# B&R Automation Studio project mappCnc
Automation Studio 4.12.11.2 SP; technology packages: mappCockpit 5.24.4, mappMotion 5.31.3, mappView 5.24.8

## Configuration Config1

CPU X20CP3585, AutomationRuntime U4.93, Build 4.1.2, Safety 0.0, Vc V4.73.5

CPU X20CP3684, AutomationRuntime 6.7.6, Build 11.3.0, Vc 6.7.0

### Task classes (Cpu.sw)
```
Cyclic#1:
  Cnc <- Motion.Cnc.prg
Cyclic#4 (cycle 200000 us, tolerance 200000 us):
  Draw <- Visualization.Draw.prg
DataObjects: McAcpSys
NcDataObjects: McDriveLog, World <- Motion.World.dob
VcDataObjects: Visu <- Visualization.Visu.dob
Binaries: arsvcreg, udbdef, McAcpDrv, McMechSys, McAcpSim, TCData, vcchspot, vcfile, arial, vctcal, vccbmp, vccstr, vcbclass, mCoWebSc, vcgclass, vcdsint, vcnet, vcmgr, arflatprv, Visu03, vcshared, vcrt, vcpdvnc, arcoal, vcpdsw, visvc, vcpfar00, vcctext, Visu01, vcfntttf, vcalarm, vcpkat, Visu02, vcdsloc, mvLoader, Role, iomap, Config_2, Hierarchy, Config_3, arconfig, asfw, sysconf, Config_4, User, ashwac, Config_1, ashwd, TraceConfi, Settings
Libraries: McBase, McAxGroup, McPathGen, McAxis, McProgInt, McAcpAx, MpCnc, MpBase, MpAxis, visapi, CoTrace, AsZip, FileIO, runtime, MpWebXs, AsArSdm, powerlnk, asarlog, asieccon, asmem, brsystem, astime, sys_lib, asarprof, dataobj, vcresman, arssl, asio, asepl
```

### Task classes (Cpu.sw)
```
Cyclic#1:
  Cnc <- Motion.Cnc.prg
Cyclic#4 (cycle 200000 us, tolerance 200000 us):
  Draw <- Visualization.Draw.prg
DataObjects: McAcpSys
NcDataObjects: McDriveLog, World <- Motion.World.dob
VcDataObjects: Visu <- Visualization.Visu.dob
Binaries: arsvcreg, udbdef, McAcpDrv, McMechSys, McAcpSim, TCData, vcchspot, vcfile, arial, vctcal, vccbmp, vccstr, vcbclass, mCoWebSc, vcgclass, vcdsint, vcnet, vcmgr, arflatprv, Visu03, vcshared, vcrt, vcpdvnc, arcoal, vcpdsw, visvc, vcpfar00, vcctext, Visu01, vcfntttf, vcalarm, vcpkat, Visu02, vcdsloc, mvLoader, Role, iomap, Config_2, Hierarchy, Config_3, arconfig, asfw, sysconf, Config_4, User, ashwac, Config_1, ashwd, TraceConfi, Settings
Libraries: visapi, AsZip, FileIO, runtime, AsArSdm, powerlnk, asarlog, asieccon, asmem, brsystem, astime, sys_lib, asarprof, dataobj, vcresman, arssl, asio, asepl, McBase, MpBase, McAxGroup, McAcpAx, McAxis, McPathGen, MpAxis, McProgInt, MpCnc, CoTrace
```

### Hardware
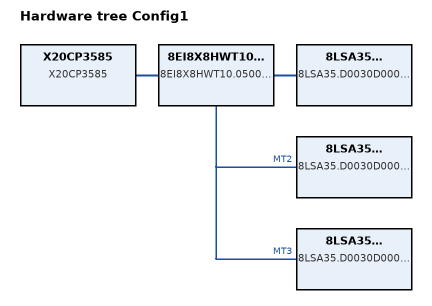
```
8EI8X8HWT10.0500-1 : 8EI8X8HWT10.0500-1 v2.4.0.0  [PLK1 -> X20CP3585.IF3 [Cable Type=PowerlinkCable, Length=10, Version=1.0.0.3]; MT2 -> 8LSA35.D0030D000-0a.MT; MT3 -> 8LSA35.D0030D000-0b.MT]
  DriveConfiguration/Module:
    McAcoposTypeID = AcoposP3TConfig
    ActivateACOPOSSimulationOnPLC = 0
  DriveConfiguration/Channel[1]/RealAxis:
    AxisReference = gAxisQX
    MechanicalElementsIsInvisible = 0
  DriveConfiguration/Channel[1]/RealAxis/MechanicalElements/Gearbox:
    InputIsReadOnly = 0
    Input = 1
    OutputIsReadOnly = 0
    Output = 1
  DriveConfiguration/Channel[1]/RealAxis/MechanicalElements/RotaryToLinearTransformation:
    ReferenceDistanceIsReadOnly = 0
    ReferenceDistance = 1
  DriveConfiguration/Channel[1]/RealAxis/EncoderLink:
    ParameterSetSelection = Automatic
  DriveConfiguration/Channel[1]/RealAxis/Controller:
    ModeIsReadOnly = 0
    Mode = PositionController
  DriveConfiguration/Channel[1]/RealAxis/Controller/Mode/Position:
    ProportionalGain = 50.0
    IntegrationTime = 0.0
    PredictionTime = 0.0004
    TotalDelayTime = 0.0004
  DriveConfiguration/Channel[1]/RealAxis/Controller/Mode/Speed:
    ProportionalGainIsReadOnly = 0
    ProportionalGain = 2.0
    IntegrationTimeIsReadOnly = 0
    IntegrationTime = 0.0
    FilterTimeIsReadOnly = 0
    FilterTime = 0.0
  DriveConfiguration/Channel[1]/RealAxis/Controller/Mode/LoopFilters:
    LoopFilterXIsReadOnly = 0
    LoopFilter1 = NotUsed
    LoopFilter2 = NotUsed
    LoopFilter3 = NotUsed
  DriveConfiguration/Channel[1]/RealAxis/Homing:
    ModeIsReadOnly = 0
    Mode = Direct
  DriveConfiguration/Channel[1]/RealAxis/Homing/Mode:
    Position = 0.0
    ReferencePulse = NotUsed
  DriveConfiguration/Channel[1]/RealAxis/Homing:
    RestorePositionVariable = 
  DriveConfiguration/Channel[1]/RealAxis/StopReaction:
    QuickstopIsReadOnly = 0
    Quickstop = DecelerationLimit
    DriveErrorIsReadOnly = 0
    DriveError = DecelerationLimit
  DriveConfiguration/Channel[1]/RealAxis/MovementErrorLimits:
    PositionError = 1.0
    VelocityErrorMonitoring = Automatic1
  DriveConfiguration/Channel[1]/RealAxis:
    JerkFilterIsReadOnly = 0
    JerkFilter = NotUsed
    ZeroVibrationFilter = NotUsed
  DriveConfiguration/Channel[1]/RealAxis/DigitalInputs/HomingSwitch:
    SourceIsReadOnly = 0
    Source = NotUsed
    Level = High
  DriveConfiguration/Channel[1]/RealAxis/DigitalInputs/PositiveLimitSwitch:
    SourceIsReadOnly = 0
    Source = NotUsed
    Level = High
  DriveConfiguration/Channel[1]/RealAxis/DigitalInputs/NegativeLimitSwitch:
    SourceIsReadOnly = 0
    Source = NotUsed
    Level = High
  DriveConfiguration/Channel[1]/RealAxis/DigitalInputs/Trigger1:
    Source = X8Trigger1
    Level = High
  DriveConfiguration/Channel[1]/RealAxis/DigitalInputs/Trigger2:
    Source = X8Trigger2
    Level = High
  DriveConfiguration/Channel[1]/RealAxis/DigitalInputs/Quickstop:
    Input = Trigger2
  DriveConfiguration/Channel[1]/RealAxis/Simulation:
    SimulationModeOnPLC = SetValueGeneration
    SimulationModeOnACOPOS = NotUsed
  DriveConfiguration/Channel[1]:
    ExternalEncoderAxis = NotUsed
  DriveConfiguration/Channel[2]/RealAxis:
    AxisReference = gAxisQY
    MechanicalElementsIsInvisible = 0
  DriveConfiguration/Channel[2]/RealAxis/MechanicalElements/Gearbox:
    InputIsReadOnly = 0
    Input = 1
    OutputIsReadOnly = 0
    Output = 1
  DriveConfiguration/Channel[2]/RealAxis/MechanicalElements/RotaryToLinearTransformation:
    ReferenceDistanceIsReadOnly = 0
    ReferenceDistance = 1
  DriveConfiguration/Channel[2]/RealAxis/EncoderLink:
    ParameterSetSelection = Automatic
  DriveConfiguration/Channel[2]/RealAxis/Controller:
    ModeIsReadOnly = 0
    Mode = PositionController
  DriveConfiguration/Channel[2]/RealAxis/Controller/Mode/Position:
    ProportionalGain = 50.0
    IntegrationTime = 0.0
    PredictionTime = 0.0004
    TotalDelayTime = 0.0004
  DriveConfiguration/Channel[2]/RealAxis/Controller/Mode/Speed:
    ProportionalGainIsReadOnly = 0
    ProportionalGain = 2.0
    IntegrationTimeIsReadOnly = 0
    IntegrationTime = 0.0
    FilterTimeIsReadOnly = 0
    FilterTime = 0.0
  DriveConfiguration/Channel[2]/RealAxis/Controller/Mode/LoopFilters:
    LoopFilterXIsReadOnly = 0
    LoopFilter1 = NotUsed
    LoopFilter2 = NotUsed
    LoopFilter3 = NotUsed
  DriveConfiguration/Channel[2]/RealAxis/Homing:
    ModeIsReadOnly = 0
    Mode = Direct
  DriveConfiguration/Channel[2]/RealAxis/Homing/Mode:
    Position = 0.0
    ReferencePulse = NotUsed
  DriveConfiguration/Channel[2]/RealAxis/Homing:
    RestorePositionVariable = 
  DriveConfiguration/Channel[2]/RealAxis/StopReaction:
    QuickstopIsReadOnly = 0
    Quickstop = DecelerationLimit
    DriveErrorIsReadOnly = 0
    DriveError = DecelerationLimit
  DriveConfiguration/Channel[2]/RealAxis/MovementErrorLimits:
    PositionError = 1.0
    VelocityErrorMonitoring = Automatic1
  DriveConfiguration/Channel[2]/RealAxis:
    JerkFilterIsReadOnly = 0
    JerkFilter = NotUsed
    ZeroVibrationFilter = NotUsed
  DriveConfiguration/Channel[2]/RealAxis/DigitalInputs/HomingSwitch:
    SourceIsReadOnly = 0
    Source = NotUsed
    Level = High
  DriveConfiguration/Channel[2]/RealAxis/DigitalInputs/PositiveLimitSwitch:
    SourceIsReadOnly = 0
    Source = NotUsed
    Level = High
  DriveConfiguration/Channel[2]/RealAxis/DigitalInputs/NegativeLimitSwitch:
    SourceIsReadOnly = 0
    Source = NotUsed
    Level = High
  DriveConfiguration/Channel[2]/RealAxis/DigitalInputs/Trigger1:
    Source = X8Trigger1
    Level = High
  DriveConfiguration/Channel[2]/RealAxis/DigitalInputs/Trigger2:
    Source = X8Trigger2
    Level = High
  DriveConfiguration/Channel[2]/RealAxis/DigitalInputs/Quickstop:
    Input = Trigger2
  DriveConfiguration/Channel[2]/RealAxis/Simulation:
    SimulationModeOnPLC = SetValueGeneration
    SimulationModeOnACOPOS = NotUsed
  DriveConfiguration/Channel[2]:
    ExternalEncoderAxis = NotUsed
  DriveConfiguration/Channel[3]/RealAxis:
    AxisReference = 
    MechanicalElementsIsInvisible = 0
  DriveConfiguration/Channel[3]/RealAxis/MechanicalElements/Gearbox:
    InputIsReadOnly = 0
    Input = 1
    OutputIsReadOnly = 0
    Output = 1
  DriveConfiguration/Channel[3]/RealAxis/MechanicalElements/RotaryToLinearTransformation:
    ReferenceDistanceIsReadOnly = 0
    ReferenceDistance = 1
  DriveConfiguration/Channel[3]/RealAxis/EncoderLink:
    ParameterSetSelection = Automatic
  DriveConfiguration/Channel[3]/RealAxis/Controller:
    ModeIsReadOnly = 0
    Mode = PositionController
  DriveConfiguration/Channel[3]/RealAxis/Controller/Mode/Position:
    ProportionalGain = 50.0
    IntegrationTime = 0.0
    PredictionTime = 0.0004
    TotalDelayTime = 0.0004
  DriveConfiguration/Channel[3]/RealAxis/Controller/Mode/Speed:
    ProportionalGainIsReadOnly = 0
    ProportionalGain = 2.0
    IntegrationTimeIsReadOnly = 0
    IntegrationTime = 0.0
    FilterTimeIsReadOnly = 0
    FilterTime = 0.0
  DriveConfiguration/Channel[3]/RealAxis/Controller/Mode/LoopFilters:
    LoopFilterXIsReadOnly = 0
    LoopFilter1 = NotUsed
    LoopFilter2 = NotUsed
    LoopFilter3 = NotUsed
  DriveConfiguration/Channel[3]/RealAxis/Homing:
    ModeIsReadOnly = 0
    Mode = Direct
  DriveConfiguration/Channel[3]/RealAxis/Homing/Mode:
    Position = 0.0
    ReferencePulse = NotUsed
  DriveConfiguration/Channel[3]/RealAxis/Homing:
    RestorePositionVariable = 
  DriveConfiguration/Channel[3]/RealAxis/StopReaction:
    QuickstopIsReadOnly = 0
    Quickstop = DecelerationLimit
    DriveErrorIsReadOnly = 0
    DriveError = DecelerationLimit
  DriveConfiguration/Channel[3]/RealAxis/MovementErrorLimits:
    PositionError = 1.0
    VelocityErrorMonitoring = Automatic1
  DriveConfiguration/Channel[3]/RealAxis:
    JerkFilterIsReadOnly = 0
    JerkFilter = NotUsed
    ZeroVibrationFilter = NotUsed
  DriveConfiguration/Channel[3]/RealAxis/DigitalInputs/HomingSwitch:
    SourceIsReadOnly = 0
    Source = NotUsed
    Level = High
  DriveConfiguration/Channel[3]/RealAxis/DigitalInputs/PositiveLimitSwitch:
    SourceIsReadOnly = 0
    Source = NotUsed
    Level = High
  DriveConfiguration/Channel[3]/RealAxis/DigitalInputs/NegativeLimitSwitch:
    SourceIsReadOnly = 0
    Source = NotUsed
    Level = High
  DriveConfiguration/Channel[3]/RealAxis/DigitalInputs/Trigger1:
    Source = X8Trigger1
    Level = High
  DriveConfiguration/Channel[3]/RealAxis/DigitalInputs/Trigger2:
    Source = X8Trigger2
    Level = High
  DriveConfiguration/Channel[3]/RealAxis/DigitalInputs/Quickstop:
    Input = Trigger2
  DriveConfiguration/Channel[3]/RealAxis/Simulation:
    SimulationModeOnPLC = SetValueGeneration
    SimulationModeOnACOPOS = NotUsed
  DriveConfiguration/Channel[3]:
    ExternalEncoderAxis = NotUsed
8LSA35.D0030D000-0 : 8LSA35.D0030D000-0 v1.0.5.40  [MT -> 8EI8X8HWT10.0500-1.MT1]
8LSA35.D0030D000-0a : 8LSA35.D0030D000-0 v1.0.5.40  [MT -> 8EI8X8HWT10.0500-1.MT2]
8LSA35.D0030D000-0b : 8LSA35.D0030D000-0 v1.0.5.40  [MT -> 8EI8X8HWT10.0500-1.MT3]
X20CP3585 : X20CP3585 v1.13.0.0
  Connector IF2:
    ActivateDevice = 1
    ActivateIna = 0
    Vnc1
    VncVcObjectName1 = Visu
    VncKeyMappingFile1 = VC\PS2-Keyboard.dis
  Connector IF3:
    DNAConfiguration = manual
    Channel1
    ChannelID1 = McAcpBroadcast
    ChannelType1 = OCTET[24]
  ConfigurationID = mappCnc_Config1
  UserPartitionSize = 0
  Simulation = 1
  TimerDeviceType = EPLX2X
  TimerDevice = X20CP3585.IF3
  TaskClassIdleTime = 4000
  CyclicTaskClassCount = 4
  Cyclic1Tolerance = 0
  Cyclic1Output = 1
  Cyclic4Duration = 200000
  Cyclic4Tolerance = 200000
  FileDevice1
  FileDeviceName1 = CNC_PrgDir
  FileDevicePath1 = C:\Temp
  FileDevice2
  FileDeviceName2 = mappCockpitDir
  FileDevicePath2 = C:\Temp
  ActivateOpcUa = 1
  OpcUaInformationModels_PV_Version = 1
```

### Config_1.axesgroup - X20CP3585/mappMotion/3AxesCNCXYZ/Config_1.axesgroup
```
Element gCncXYZ (Type=axesgroup)
  Type = PathGenAxesGroup
    ProcessingTaskClass = 1
    License = 1
    PhysicalAxes:
      JointAxes:
        JointAxis[1]:
          Name = QX
          AxisRef = gAxisQX
        JointAxis[2]:
          Name = QY
          AxisRef = gAxisQY
        JointAxis[3]:
          Name = QZ
          AxisRef = gAxisQZ
    MechanicalSystem:
      MechSysRef = MechSys_3AxCNCXYZ
    BasicSettings:
      ModalDataBehaviour = ResetToDefault
      GeometryPlanning:
        MaxCornerDeviation = 0.0
        MaxTangentialTransitionDeviation = 0.0
        MaxRadiusDeviation = 0.001
        WorkingPlane = XY
      TrajectoryPlanning = Basic
        LimitCheckResolution = UserDefinedTime
          Time = 0.01
        BufferTime = UserDefinedTime
          Time = 0.1
    AxesGroupFeatures:
      FeatureRef[1] = GCode
      FeatureRef[2] = M-Functions
```

### Config_2.axis - X20CP3585/mappMotion/3AxesCNCXYZ/Config_2.axis
```
Element gAxisQX (Type=axis)
  BaseType = LinearBounded
    MeasurementUnit = 5066068
    MeasurementResolution = 0.01
    CountDirection = Standard
  MovementLimits = Internal
    Position:
      LowerLimit = -1000.0
      UpperLimit = 1000.0
    Velocity:
      Velocity = 10.0
    Acceleration:
      Acceleration = 50.0
    Deceleration:
      Deceleration = 50.0
Element gAxisQY (Type=axis)
  BaseType = LinearBounded
    MeasurementUnit = 5066068
    MeasurementResolution = 0.01
    CountDirection = Standard
  MovementLimits = Internal
    Position:
      LowerLimit = -1000.0
      UpperLimit = 1000.0
    Velocity:
      Velocity = 10.0
    Acceleration:
      Acceleration = 50.0
    Deceleration:
      Deceleration = 50.0
Element gAxisQZ (Type=axis)
  BaseType = LinearBounded
    MeasurementUnit = 5066068
    MeasurementResolution = 0.01
    CountDirection = Standard
  MovementLimits = Internal
    Position:
      LowerLimit = -1000.0
      UpperLimit = 1000.0
    Velocity:
      Velocity = 10.0
    Acceleration:
      Acceleration = 50.0
    Deceleration:
      Deceleration = 50.0
```

### Config_4.axesgroupfeature - X20CP3585/mappMotion/3AxesCNCXYZ/Config_4.axesgroupfeature
```
Element GCode (Type=axesgroupfeature)
  Type = Program
    DefaultLanguage = BRGCode
    Location = Default
      FileDevice = CNC_PrgDir
Element M-Functions (Type=axesgroupfeature)
  Type = MFunctions
    MFunction[1]:
      IndexType = Single
        Index = 7
      Blocking = Enabled
      Output = Before
      InSimulation = NotUsed
      PvMapping = ::Cnc:MFunc_CutterDown
    MFunction[2]:
      IndexType = Single
        Index = 8
      Blocking = Enabled
      Output = Before
      InSimulation = NotUsed
      PvMapping = ::Cnc:MFunc_CutterUp
```

### Config_1.axesgroup - X20CP3684/mappMotion/3AxesCNCXYZ/Config_1.axesgroup
```
Element gCncXYZ (Type=axesgroup)
  Type = PathGenAxesGroup
    ProcessingTaskClass = 1
    License = 1
    PhysicalAxes:
      JointAxes:
        JointAxisAxisRefIsReadOnly = 0
        JointAxis[1]:
          Name = QX
          AxisRef = gAxisQX
        JointAxis[2]:
          Name = QY
          AxisRef = gAxisQY
    MechanicalSystem:
      MechSysRefIsReadOnly = 0
      MechSysRef = MechSys
    BasicSettings:
      ModalDataBehaviour = ResetToDefault
      GeometryPlanning:
        TCPResolutionIsReadOnly = 0
        TCPResolution:
          LengthResolution = 0.001
          AngleResolution = 0.001
        Rounding:
          PathDistance = 0.0
          SymmetricRounding = Yes
          LastSegment = Half
          AvoidZeroCurvature = No
        RoundingMode = Standard
        MaxCornerDeviation = 0.0
        MaxTangentialTransitionDeviation = 0.0
        MaxRadiusDeviation = 0.1
        WorkingPlane = XY
      TrajectoryPlanningIsReadOnly = 0
      TrajectoryPlanning = Basic
        LimitCheckResolutionIsReadOnly = 0
        LimitCheckResolution = UserDefinedTime
          TimeIsReadOnly = 0
          Time = 0.01
        BufferTime = UserDefinedTime
          Time = 0.1
        BarrierParametrization = JointCoordinates
        TorqueLimitConsideration = Exact
      Miscellaneous:
        NonMovementsLimit = NotUsed
        TimeStretchOverride:
          JerkSuppression = NotUsed
    StopReaction:
      AxisError:
        AxisReactionIsReadOnly = 0
    AxesGroupFeatures:
      FeatureRef[1] = GCode
      FeatureRef[2] = M-Functions
      FeatureRef[3] = Path-Definition
  Alarms = None
```

### Config_2.axis - X20CP3684/mappMotion/3AxesCNCXYZ/Config_2.axis
```
Element gAxisQX (Type=axis)
  BaseTypeIsReadOnly = 0
  BaseType = LinearBounded
    MeasurementUnit = 5066068
    MeasurementResolutionIsReadOnly = 0
    MeasurementResolution = 0.01
    CountDirectionIsReadOnly = 0
    CountDirection = Standard
  MovementLimitsIsReadOnly = 0
  MovementLimits = Internal
    Position:
      LowerLimitMin = -1.79769313486231E308
      UpperLimitMax = 1.79769313486231E308
      LowerLimit = -2000
      UpperLimit = 2000
    VelocityIsReadOnly = 0
    Velocity:
      VelocityMax = 3.4E38
      Velocity = 500
    AccelerationIsReadOnly = 0
    Acceleration:
      AccelerationMax = 3.4E38
      Acceleration = 500.0
    DecelerationIsReadOnly = 0
    Deceleration:
      DecelerationMax = 3.4E38
      Deceleration = 500.0
  Alarms = None
Element gAxisQY (Type=axis)
  BaseTypeIsReadOnly = 0
  BaseType = LinearBounded
    MeasurementUnit = 5066068
    MeasurementResolutionIsReadOnly = 0
    MeasurementResolution = 0.01
    CountDirectionIsReadOnly = 0
    CountDirection = Standard
  MovementLimitsIsReadOnly = 0
  MovementLimits = Internal
    Position:
      LowerLimitMin = -1.79769313486231E308
      UpperLimitMax = 1.79769313486231E308
      LowerLimit = -2000
      UpperLimit = 2000
    VelocityIsReadOnly = 0
    Velocity:
      VelocityMax = 3.4E38
      Velocity = 500
    AccelerationIsReadOnly = 0
    Acceleration:
      AccelerationMax = 3.4E38
      Acceleration = 500.0
    DecelerationIsReadOnly = 0
    Deceleration:
      DecelerationMax = 3.4E38
      Deceleration = 500.0
  Alarms = None
```

### Config_3.mechanicalsystem - X20CP3684/mappMotion/3AxesCNCXYZ/Config_3.mechanicalsystem
```
Element MechSys (Type=mechanicalsystem)
  TypeIsReadOnly = 0
  Type = 2AxesCNC
    Subtype = 2AxesCNCXY
      CoordinatesNames = Default
        XCoordinateName = X
        YCoordinateName = Y
      WireFrameModel = Standard
        FlangeToTcp = ConnectionLine
          DistanceMin = -1.79769313486231E308
          DistanceMax = 1.79769313486231E308
          Distance = 0.0
      JointAxesPositionLimits:
        JointAxisIsReadOnly = 0
        JointAxis[1] = UseAxisLimits
        JointAxis[2] = UseAxisLimits
```

### Config_4.axesgroupfeature - X20CP3684/mappMotion/3AxesCNCXYZ/Config_4.axesgroupfeature
```
Element GCode (Type=axesgroupfeature)
  Type = Program
    ModalDataBehaviour = UseAxesGroupSettings
    InitialSettings:
      InterpolationTypes = LinearRapid
      PositionCoordinates = Absolute
      CircleCoordinates = Relative
      JACS_ACSProgramming = JACS
      ContourConnection = Inactive
      AccuracyHoldDelays = None
      ProgrammingUnits = UseAxesGroupSettings
      Feedrates:
        FeedPath = Standard
        FeedCharacteristic = StandardCharacteristic
        FeedType = Feedrate
        FeedReduction = Inactive
        FeedrateValue = 0.0
        InverseFeedrateValue = 0.0
        FeedratePerRevValue = 0.0
    DefaultLanguage = BRGCode
    Location = Default
      FileDevice = CNC_PrgDir
Element M-Functions (Type=axesgroupfeature)
  Type = MFunctions
    ModalDataBehaviour = UseAxesGroupSettings
    MFunction[1]:
      IndexType = Single
        Index = 7
      Blocking = Enabled
      Output = Before
      InSimulation = NotUsed
      PvMapping = ::gMFunc_CutterDown
      Counter
    MFunction[2]:
      IndexType = Single
        Index = 8
      Blocking = Enabled
      Output = Before
      InSimulation = NotUsed
      PvMapping = ::gMFunc_CutterUp
      Counter
Element Path-Definition (Type=axesgroupfeature)
  Type = PathDefinitions
    ModalDataBehaviour = UseAxesGroupSettings
    PathDefinition[1]:
      Name = Path1
      Type = PhysicalAxes
      Limit = Internal
        Velocity = NotUsed
        Acceleration = NotUsed
        Deceleration = NotUsed
        Jerk = NotUsed
```

## Logical view

Binary libraries used (declarations not repeated): operator, runtime, astime, AsIecCon, visapi, AsZip, FileIO, AsArSdm, MpBase, MpWebXs 5.24.7, CoTrace 5.02.3, McBase 5.31.3, McPathGen 5.31.3, MpAxis 5.31.3, McAcpAx 5.31.3, McAxis 5.31.3, McProgInt 5.31.3, McAxGroup 5.31.3, MpCnc 5.31.3

### Package Logical/Libraries - Globale Bibliotheken

### Motion.var
```iecst
VAR
	g_positionY : LREAL;
	gMFunc_CutterDown : BOOL;
	gMFunc_CutterUp : BOOL;
	g_positionX : LREAL;
END_VAR
```

### Program Logical/Motion/Cnc (IEC)

#### Variables.var
```iecst
VAR
	fbMpCnc : MpCnc2Axis;
	CncParameters : MpCnc4AxisParType;
END_VAR
```

#### Cyclic.st
```iecst
PROGRAM _CYCLIC
	fbMpCnc();

	g_positionX := fbMpCnc.X;
	g_positionY := fbMpCnc.Y;

END_PROGRAM
```

#### Exit.st
```iecst
PROGRAM _EXIT
	fbMpCnc.Enable := FALSE;
    fbMpCnc.Power  := FALSE;
    fbMpCnc.Home   := FALSE;
    fbMpCnc();

END_PROGRAM
```

#### Init.st
```iecst
PROGRAM _INIT
	fbMpCnc.MpLink := ADR(gCncXYZ);
	fbMpCnc.Enable := TRUE;
	fbMpCnc.Parameters := ADR(CncParameters);

	fbMpCnc.Override := 100.0;

	CncParameters.ProgramName := 'World';

END_PROGRAM
```

### Data object Logical/Motion/World (Cnc)

#### CncProg.cnc - CNC program (G-Code)
```
F10000
G90
G0 X200 Y0
G91
G1 X81 Y474.3
M7
X-9 Y-0.4
X-1.9 Y-2.4
X-6.5 Y-12.8
X-8.7 Y-20.2
X-3.9 Y-11.1
X-0.2 Y-3
X0.8 Y-1.9
X1.6 Y-1.2
X2.1 Y-0.1
X2.8 Y2.9
X2 Y4.7
X0.7 Y1.9
X1.8 Y1.1
X3 Y-0.3
X2.9 Y-0.8
X0.9 Y0.4
X0.6 Y0.9
X-0.2 Y3
X-0.9 Y5
X0.8 Y1.8
X4.7 Y2.1
X2.9 Y-0.7
X9.4 Y-4
X3.9 Y-1.4
X3.8 Y-1.4
X4.9 Y-4
X8.2 Y-2.2
X3.1 Y0.7
X3.6 Y2.2
G3 X-1.2 Y3.7 I-1.1 J1.7
G1 X-5.3 Y0.2
X-3 Y1
X-3 Y0.7
X-5.1 Y3.5
X-9.8 Y4
X-2.6 Y1.7
X-5 Y1.3
X-5.1 Y3.3
X-1.6 Y2.7
X-0.2 Y2
X1 Y1.8
X2.9 Y0.9
X5.3 Y-0.1
X6.4 Y1.1
X2.9 Y-0.8
X6.6 Y-3.5
X1.7 Y-2.5
X1.6 Y-2.6
X1.9 Y-0.6
X1 Y0.4
X0.6 Y2
X-0.9 Y3
X-3.4 Y5.5
X-2.2 Y7.3
X-0.5 Y6.4
X-2.1 Y3.7
X-2.8 Y4.5
X-1.5 Y4
X-3 Y2.7
X-3 Y1.3
X-2 Y-0.2
X-2.4 Y-1.9
X-8.6 Y-14.3
X0.2 Y-1.4
M8
G0 X170.7 Y0.7
M7
G1 X0 Y-5
X1.7 Y-2.5
X3.9 Y-3.4
X2.5 Y-3.1
X3.1 Y0
X3 Y0.4
X5.8 Y-2.3
X4.1 Y-0.3
X2 Y0.7
X1.3 Y1.6
X0.4 Y4.1
X-1.3 Y4
X-2.8 Y4.4
X-2.8 Y1.5
X-3 Y-0.2
X-5.2 Y-1
X-2.9 Y1.2
X-6 Y5.7
X-6.5 Y3
X-2.7 Y1.7
X-2.1 Y0.3
X-1.7 Y-1.1
X-2.2 Y-3.6
X-3.7 Y-3.7
X-1 Y-5.2
X0.7 Y-3
X1.5 Y-1.5
X2 Y0.3
X2.1 Y2.3
X2.7 Y1.3
X2.1 Y0.2
X2.9 Y-1.3
X0.9 Y-0.6
X1.2 Y0.1
M8
G0 X3.7 Y67.3
M7
G1 X-10.3 Y4.1
G3 X-3.7 Y-8.8 I0.9 J-5.6
G1 X3.5 Y-3.8
X0.7 Y-1.9
X-1.3 Y-1.6
X-4.1 Y-1.1
X-1.3 Y-1.5
X-0.3 Y-3.2
X0.7 Y-1.9
X1.6 Y-1.3
X5.8 Y-2.2
X2.4 Y-1.9
X1.9 Y-3.7
X1.6 Y-3.8
G3 X9.9 Y1.3 I4.7 J2.8
G1 X0.3 Y5.1
X-1.5 Y7.1
X-2 Y7
X0.3 Y3.1
X2.3 Y6.9
X0.9 Y4
X-2 Y4.8
X-2.5 Y1.9
X-3.1 Y0.3
X-8.7 Y-3.2
X-1.4 Y-1.6
M8
G0 X-187.6 Y452
M7
G1 X-7.6 Y-5
X-1.5 Y-7.2
X-0.1 Y-4.1
X-0.9 Y-7.2
X0.8 Y-4.1
X-0.1 Y-3.1
X0.3 Y-0.9
X1.9 Y-0.9
X2.9 Y0.9
X3.9 Y3.4
X2 Y0.4
X1.9 Y-0.7
X4.4 Y-2.9
X1.1 Y-2.9
X0.8 Y-3.1
X1.5 Y-1.4
X3 Y-0.3
X5.1 Y0.3
X6.9 Y2
X2.1 Y2.2
X0.3 Y2
X-1 Y1.8
X-10.9 Y10.9
X-3.5 Y2.2
X-1.6 Y2.6
X-0.6 Y4.1
X0.5 Y4.1
X-0.2 Y4.2
X1 Y4.1
X0.2 Y4.1
X-0.8 Y4.1
X2.1 Y6.9
X-0.6 Y2.9
X-4.1 Y3.2
X-2.7 Y1.7
X-4.3 Y4.5
X-2 Y0.7
X-1 Y-0.1
X-1.5 Y-1.4
X-2.1 Y-7.1
X-2.5 Y-13.3
X-1.8 Y-4.9
X-1.3 Y-2.9
X0.7 Y-3
X1.7 Y-1.8
M8
G0 X535.1 Y154.3
M7
G1 X0.4 Y21.4
X-3.4 Y4.4
X-17.8 Y17.2
X-13.3 Y11.8
X-18.6 Y14.2
X-12.7 Y8.7
X-17.5 Y10.3
X-19.8 Y9.3
X-27.8 Y10.6
X-27.9 Y8.7
X-25.4 Y5.6
X-15.3 Y2.3
X-19.5 Y1.2
X-21.4 Y-0.7
X-23.9 Y-2.6
X-22.1 Y-3.8
X-20.2 Y-5
X-27 Y-8.3
X-21.3 Y-9
X-20.1 Y-10.5
X-28 Y-17.4
X-10.6 Y-7.3
X-18.9 Y-15.8
X-18.3 Y-17.8
X-13.6 Y-15.2
X-16.5 Y-21.3
X-0.4 Y-2
X0.2 Y-1
X1.9 Y-0.9
X3.1 Y0.1
X5 Y0.7
X5.1 Y-0.7
X5.9 Y-1.8
X8.1 Y-6.5
X3.1 Y-0.5
X1.9 Y0.7
X6.6 Y6.5
X4.1 Y9.3
X1.8 Y7
X1.5 Y2.6
X0.8 Y0.7
X1 Y0.2
X0.9 Y-0.5
X0.6 Y-2
X-3 Y-8
X-0.9 Y-6.5
X-4.2 Y-8.2
X-5 Y-10
X-5.2 Y-7.6
X-3.4 Y-8
X-1.1 Y-1.9
X-7 Y-6.8
X-1 Y-3.1
X-0.7 Y-6.5
X1.3 Y-2.9
X5 Y-4
X2.5 Y-3.5
X2.7 Y-5.7
X4.2 Y-4.4
X7.5 Y-3.9
X9.7 Y-2.1
X5.4 Y-0.2
X10.3 Y-1.3
X5.3 Y-1.7
X10.3 Y-5.4
X2.1 Y-0.4
X8.3 Y2.4
X3 Y-0.6
X7.4 Y-4.2
X5 Y-1.9
X4.3 Y-0.3
X7.4 Y1.3
X12.8 Y5.3
X9.6 Y2.6
X10.7 Y0.5
X6.3 Y-0.9
X9.2 Y-1.6
X9 Y-3.8
X5.6 Y-6.1
X4.5 Y-2.8
X9.3 Y-2.9
X10.3 Y-1.9
X5.8 Y-4.4
X9.3 Y-4.4
X1.6 Y-1.3
X0.4 Y-1
X-0.2 Y-1
X-0.8 Y-0.6
X-2.1 Y0.2
X-8.2 Y4
X-7.1 Y1.3
X-2.9 Y0.9
X-1.5 Y-1.3
X-0.1 Y-2
X0.9 Y-2
X2.6 Y-1.7
X7.9 Y-3.3
X4 Y-1.5
X9.3 Y-7
X3.9 Y-1.4
X3.4 Y0
X4.2 Y0.6
X5.2 Y-1.7
X3.4 Y-4
X4.3 Y-8.2
X3.6 Y-8.8
X1.5 Y-5.2
X0.3 Y-3.1
X-1 Y-5.5
X0.5 Y-2.2
X2.9 Y-4.1
X2.6 Y-3.3
X4.2 Y-8.4
X5.2 Y-7.7
X2.8 Y-1.6
X2.7 Y-1.6
X7 Y-8.2
X2 Y-4.8
X-0.6 Y-5.4
X-0.8 Y-3
X0.6 Y-2.1
X2.1 Y-2.3
X2.6 Y-1.8
X7.2 Y-2.5
X3.2 Y-0.1
X3.8 Y1.6
X2.9 Y2.9
X2.7 Y3.1
X3.8 Y1.9
X6.4 Y1.5
X2 Y-0.5
X1.7 Y-1.3
X2.2 Y-0.3
X5.2 Y1.1
X3 Y-0.7
X1.6 Y-1.3
X2.2 Y-3.7
X5.3 Y-3.5
X2.3 Y-2.2
X4.8 Y-2.3
X7.1 Y-6.3
X4.6 Y-2.6
X4.4 Y-4.4
X1.5 Y-2.9
X1.7 Y-5.1
X3.3 Y-5.5
X2.7 Y-3.2
X3.9 Y-2
X5.1 Y-1
X9.7 Y0.4
X10.3 Y-1.6
X10.6 Y0.6
X8.5 Y-0.8
X8.3 Y-1.7
X5.3 Y0.3
X7.2 Y1.5
X5.2 Y0
X9.3 Y-3
X5.1 Y0.1
X4.7 Y-2.4
X3.7 Y-1.9
X5.2 Y-0.7
X6 Y1.6
X5.3 Y1.3
X2.1 Y-0.2
X17.5 Y-7.4
X9.9 Y-5.1
X3.1 Y-4.2
X2.8 Y-5.5
X2.3 Y-3.5
X1.2 Y-6
X-0.9 Y-7
X-1.4 Y-2.7
X-1.7 Y-0.9
X-1.7 Y1.2
X-2.7 Y4.3
X-4.1 Y4.5
X-6.7 Y4.6
X-3.1 Y0.2
X-7.1 Y-2.1
X-5.9 Y-2.3
X-2 Y-0.1
X-2.7 Y1.8
X-2.3 Y3.3
X-2 Y0.9
X-2 Y-0.2
X-4.4 Y-2.7
X-13.5 Y-2.2
X-3.8 Y-2
X-6 Y-1.7
X-1.6 Y-1.5
X-3.8 Y-6.8
X-1.9 Y-2.7
X-3.8 Y-1.8
X-6.3 Y-1.1
X-1.5 Y-1.4
X-2.4 Y-3.7
X-5.2 Y-3.9
X-8.7 Y-5
X-3.7 Y-2.2
X-5.1 Y-1.5
X-5.8 Y-3
X-4.4 Y0
X-4.2 Y0.5
X-2.8 Y-1.6
X-3.5 Y-2.5
X-3.7 Y-5.4
X-3 Y-3.2
X-2.1 Y-7
X-2.2 Y-2.3
X-4 Y-1.8
X-5 Y-1.8
X-7.4 Y-1.1
X-5.5 Y-0.6
X-6.5 Y0.7
X-4.1 Y-1.1
X-10.9 Y-5.6
X-7 Y-2.9
X-3 Y-1.3
X-2.2 Y-0.2
X-2.9 Y1.4
X-1.7 Y2.7
X-1.4 Y3
X-4.1 Y3.5
X-1.3 Y4
X0 Y4.3
X-0.1 Y3.2
X-1.2 Y5.1
X-3.7 Y10.2
X-2.7 Y12.1
X-2.8 Y3.3
X-7.3 Y4.9
X-3.6 Y2.3
X-3.3 Y4.2
X-1.4 Y4.2
X-0.6 Y6.4
X-0.1 Y4.2
X-1.2 Y3
X-3.5 Y2.5
X-4.4 Y9
X-3.8 Y5.2
X-0.8 Y4.1
X0.6 Y4.1
X1.3 Y3
X-0.2 Y3.2
X-1.1 Y2.9
X-1.5 Y3
X-1.7 Y9.3
X-0.6 Y4.1
X0.9 Y2.9
X1.9 Y2.5
X1 Y3.1
X3.2 Y2.7
X3.9 Y1.9
X1.6 Y2.8
X0.1 Y2.1
X-3 Y7.1
X-1.8 Y6.1
X-2.2 Y3.7
X-2.7 Y1.8
X-3.2 Y0.3
X-6.4 Y-0.7
X-1.9 Y0.9
X-1.3 Y2.8
X-1.1 Y7.2
X-0.5 Y3.2
X-1.6 Y1.5
X-2 Y0.3
X-6.1 Y-2.3
X-4.6 Y-3
X-2 Y-0.4
X-1.9 Y0.8
X-1.6 Y3.9
X-0.3 Y4.3
X1.5 Y2.7
X7.7 Y5.5
G3 X-3.4 Y17.1 I-9.8 J6.9
G1 X-3.9 Y1.8
X-4.4 Y0.4
X-5.5 Y-0.4
X-10.4 Y-2
X-4.1 Y-0.8
X-3.4 Y-2.7
X-2.8 Y-4.6
X-2.1 Y-8.1
X1 Y-9.5
X-1.1 Y-1.9
X-2.2 Y-2.4
X-1.3 Y-2.9
X0.8 Y-7.1
X2 Y-3.7
X0.7 Y-3
X2.4 Y-1.8
X4.1 Y-1.1
X7.2 Y-1.2
X1.5 Y-1.4
X0.5 Y-3.1
X-1.2 Y-1.6
X-5.4 Y-0.3
X-5.5 Y0.7
X-3.3 Y0.4
X-2.2 Y0.5
X-3.9 Y-1.2
X-2.6 Y-2.2
X-7.7 Y-12.7
X-3.3 Y-3
X-7.9 Y-3.1
X-4.6 Y-3.3
X-5.6 Y-2.8
X-4.5 Y-3.6
X-2 Y-3.6
X-1.7 Y-5
X-2.1 Y-2.7
X-4.7 Y-2.2
X-3.6 Y-1.9
X-2.3 Y-3.6
X-1.5 Y-6.2
X0.4 Y-2.1
X1.4 Y-4.1
X-2.2 Y-6.7
X-1.9 Y-3.7
X-1.9 Y-0.8
X-2 Y0.7
X-4.6 Y4.1
X-5 Y1.1
X-4.1 Y0.5
X-2.7 Y1.4
X-1 Y0
X-1.2 Y-1.7
X-0.7 Y-5.1
X-0.2 Y-9.4
X0.5 Y-3
X0.7 Y-0.8
X3 Y-0.3
X4.9 Y1.3
X1.9 Y-0.9
X1.3 Y-2.8
X1.9 Y-5.9
X0 Y-8.2
X-2.6 Y-1.6
X-3 Y0.2
X-2.8 Y1.3
X-3.3 Y2.4
X-2.9 Y1
X-10.5 Y-1.5
X-3 Y0.8
X-8.1 Y4.8
X-5.1 Y4.9
X-2.9 Y1.4
X-21.9 Y4.8
X-0.9 Y0.5
X-0.6 Y1.9
X1.5 Y3.9
X1.5 Y1.4
X2.7 Y1.6
X0.8 Y1.9
X-0.3 Y2
X-2.4 Y2
X-5.1 Y1.2
X-3.1 Y0.3
X-6.1 Y3.7
X-6.8 Y8.8
X-1.2 Y4.1
X0.7 Y2
X2.1 Y2.2
X4.8 Y2.2
X5.2 Y0.8
X5.1 Y1.5
X5.9 Y2.6
X3.1 Y-0.4
X5.1 Y-1.2
X3.2 Y0
X2.5 Y1.8
X3.1 Y4.2
X2.5 Y5.8
X4.4 Y3
X0.4 Y2.1
X-1.1 Y1.8
X-4.6 Y2.5
X-3.8 Y3.7
X-1.4 Y2.9
X-0.5 Y3.1
X-10.7 Y13.5
X-3.8 Y2.1
X-5 Y1.5
X-2.9 Y1.3
X-3.1 Y-0.5
X-3.8 Y-2.4
X-8.8 Y-8.2
X-3.8 Y-2.3
X-3.5 Y-4.6
X-3.2 Y-6.4
X-2.8 Y-6.1
X-4.6 Y-4.1
X-4.3 Y-4.6
X-3.3 Y-2.6
X-0.9 Y-3
X-0.6 Y-6.3
X-1.7 Y-2.6
X-5.3 Y-3.1
X-4.3 Y-0.6
X-3.4 Y-2.2
X-2.8 Y-1.3
X-1.4 Y-3.9
X0.5 Y-3.1
X2.3 Y-3.4
X5.9 Y-4.4
X7.6 Y-3.5
X3.1 Y0.3
X3.7 Y2.1
X2.9 Y3.1
X4.6 Y12.9
X0.7 Y0.8
X2 Y0.5
X2.9 Y-1
X1.5 Y-2.8
X0.6 Y-7.4
X2 Y-2.2
X5 Y-2
X4 Y-1.2
X1.2 Y-1.8
X1.1 Y-2.9
X3.2 Y-4.2
X0.6 Y-1.9
X-0.1 Y-1
X-3.1 Y-2.7
X-1 Y-1.8
X-2.9 Y-1.3
X-4.2 Y0
X-4.1 Y1
X-5.4 Y0
X-3.1 Y-2.7
X-3 Y-0.9
X4 Y-0.3
X2.8 Y-1.1
X1.3 Y-1.6
X0.2 Y-2
X-2 Y-3.5
X-3 Y-2.8
X-6 Y-1.6
X-4.1 Y0.3
X-2.8 Y1.3
X-4.3 Y4.5
X-3.9 Y1.2
X-6.2 Y-0.3
X-5.9 Y1.8
X-4 Y3.2
X-3.3 Y2.5
X-3.5 Y4.9
X-3.8 Y1.6
X-9.1 Y1.4
X-2.6 Y1.5
X-2.5 Y3.3
X-1.4 Y4.9
X-0.5 Y5.2
X-2.4 Y5.7
X-1.3 Y7.3
X-4.2 Y7.5
X-1.6 Y6
X-0.5 Y4.2
X-2.6 Y5.7
X0 Y4.1
X1.6 Y3.8
X2.5 Y3.2
X-0.2 Y2.1
X-5.3 Y4.6
X-0.9 Y3
X1.7 Y7.1
X1.8 Y3.7
X1 Y7.2
X-1.4 Y1.6
X-7.4 Y3.8
X-2.1 Y0.1
X-1.5 Y-1.5
X-0.6 Y-4.1
X3.5 Y-29.1
X4.5 Y-23.5
X5 Y-19.4
X7.6 Y-21.9
X9.1 Y-20.7
X10.5 Y-19.5
G3 X21 Y-5.6 I12.3 J4.1
G1 X3.2 Y-0.3
X7 Y-2.6
X2.9 Y0.7
X6 Y2.2
X10.8 Y1.8
X4.1 Y-0.2
X10.9 Y-2.4
X9.5 Y-2.4
X3.8 Y-1.4
X1.9 Y-5.7
X1.8 Y-2.6
X0.5 Y-4
X-0.6 Y-2
X-2.2 Y-2.4
X-7.9 Y-4.1
X-6.8 Y-2.4
X-8.4 Y-5.3
X-3.7 Y-4.9
X-3 Y-10.2
X-2.6 Y-3.3
X-6 Y-5.6
X-2 Y-3.6
X-5.4 Y-17.4
X-2.9 Y-4.2
X-2.6 Y-1.6
X-4 Y-1.1
X-3.1 Y-2.8
X-3.6 Y-2
X-1.4 Y-2.7
X-0.3 Y-4.1
X-0.3 Y-54.3
X0 Y-6.3
X-0.6 Y-108.9
X0.3 Y-3
X-1.7 Y-3.7
X-3.8 Y-4.9
X-0.8 Y-3
X2 Y-3.5
X1.3 Y-2.9
X1.8 Y-6.9
X1.3 Y-5.1
X5 Y-7.8
X5 Y-3.5
X1 Y0
X0.6 Y0.9
X0 Y4.3
X1.8 Y4.8
X0 Y4.2
X-0.2 Y4.3
X3.1 Y6.7
X6.2 Y6.9
X0.3 Y1
X-0.3 Y1
X-3 Y2.7
X-1.6 Y3.8
X0.6 Y1.9
X0.9 Y0.6
X3 Y-0.1
X4 Y-0.8
X2 Y0.4
X2 Y2.2
X1.3 Y1.7
X4 Y3.2
X1.8 Y1.1
X2.7 Y1.3
X0.8 Y2.9
X0.5 Y3
X0.8 Y1.9
X-0.4 Y2
X-2.6 Y1.7
X-2 Y0.1
X-1.8 Y-0.9
X-1.2 Y-1.7
X-2.6 Y-8
X-2 Y-2.2
X-2.9 Y-1.2
X-2 Y0.6
X-1.9 Y2.2
X-4.2 Y7
X-2.6 Y3.3
X-1.2 Y4
X-0.1 Y4.2
X-1 Y3
X-0.6 Y3
X-1.6 Y1.3
X-3.3 Y2.4
X-3.4 Y3.7
X-1.1 Y7.1
X0.8 Y5
X3.1 Y6.4
X2 Y2.5
X1 Y5
X4.9 Y9
X3.5 Y3.8
X1.7 Y1.1
X2.1 Y0.1
X4 Y-0.7
X7.7 Y2.7
X12.5 Y7.8
X4.2 Y4.5
X3.1 Y5.3
X2.8 Y4.3
X4.7 Y2.1
X4.1 Y0.2
X3 Y-0.5
X4.5 Y-2.4
X7 Y-1.3
X1.6 Y-1.3
X0.3 Y-3
X-0.7 Y-3
X-1.6 Y-2.6
X-1 Y-1.7
X-3.2 Y-2.5
X-1 Y-0.3
X5.2 Y-3
X8.7 Y-2.6
X2.9 Y-0.9
X1.9 Y-2.3
X-0.3 Y-4.1
X-2.2 Y-3.4
X-1.5 Y-1.3
X-9.2 Y-2.1
X-5.7 Y-2.2
X-3 Y0.2
X-5.7 Y2.2
X-4 Y-0.4
X-5.5 Y-3
X-5 Y-3.6
X-8.9 Y-2.7
G3 X-2.3 Y-8.5 I1.7 J-5
G1 X1.8 Y-0.8
X3 Y0.6
X2.6 Y1.8
X3 Y2.8
X4.8 Y2.3
X5.5 Y0.3
X4.3 Y-0.9
X2 Y-2.3
X1.7 Y-4.9
X0.6 Y-5
X-1.4 Y-4.8
X0.1 Y-1
X1.6 Y-1.2
X2 Y0.2
X0.8 Y0.6
X1.6 Y7.8
X1.2 Y1.6
X1.9 Y0.8
X4 Y0
X1.4 Y1.4
X2.8 Y4.1
X3.3 Y2.2
X3 Y0.5
X3 Y-0.4
X1.8 Y0.9
X1.8 Y2.5
X0.2 Y5
X0 Y2
X2.2 Y4.5
X1.5 Y2.6
X0.1 Y3
X-1.2 Y3.9
X0.2 Y4
X-0.8 Y1.9
X-1.7 Y1.1
X-2.9 Y-0.4
X-2.9 Y-1
X-3.1 Y0.2
X-1.7 Y1
X-0.9 Y1.8
X0.3 Y3
X2.4 Y1.8
X3 Y0.6
X3 Y-0.6
X3.8 Y-1.2
X2 Y0.6
X1 Y1.7
X2.7 Y6.6
X0.5 Y2
X1.7 Y1.1
X4.3 Y2.6
X1.2 Y2.8
X-0.8 Y1.8
X-5 Y5.1
X-4.2 Y2.7
X-4.7 Y2.1
X-5.2 Y3.1
X-6.1 Y0.7
X-3.9 Y1.4
X-1.7 Y2.6
X-0.6 Y3.1
X1.2 Y1.6
X3.6 Y2
X4.1 Y0.7
X5 Y-1.4
X0.9 Y0.4
X0.8 Y1.8
X-0.5 Y4
X2.2 Y4.5
X3.5 Y2
X6 Y1.6
X4.1 Y0.4
X1.8 Y-1.1
X0.5 Y-2
X-2.4 Y-6.7
X-2.2 Y-2.1
X-5.5 Y-2.5
X-0.5 Y-0.9
X0.3 Y-1
X2.9 Y-1
X8.1 Y0.5
X2.8 Y1.3
X1 Y-0.2
X1 Y-1.8
X0.1 Y-3.1
X-2 Y-10
X-0.1 Y-1.1
X0.4 Y-0.9
X0.9 Y-0.5
X1 Y0.2
X1.3 Y1.6
X1.9 Y3.6
X2 Y2.4
X1 Y5
X1.3 Y1.6
X1 Y0.2
X2.5 Y-1.6
X5.8 Y-5.8
X8.1 Y-1.3
X1.9 Y0.8
X1 Y1.8
X-0.3 Y10.6
X-0.5 Y6.2
X1.1 Y2.9
X2.4 Y1.9
X3.2 Y0.3
X5.2 Y0.1
X8 Y2.2
X4.1 Y-0.3
X1.4 Y-1.5
X1.1 Y-4
X2.9 Y-4.4
G2 X-14.5 Y-22.4 I-17 J-4.9
G1 X-3 Y-4.2
X-1.1 Y-1.9
X-6.3 Y-3.6
X-1.5 Y-2.8
X-0.6 Y-4.2
X0 Y-4.1
X-1.3 Y-2.7
X-2.1 Y-3.7
X0.3 Y-2.1
X2.3 Y-2.3
X6 Y-4.6
X5 Y-6.9
X3.5 Y-5.2
X1.8 Y-1
X2 Y0.4
X1.3 Y1.5
X1.5 Y4.9
X2.7 Y1.5
X1.9 Y-0.6
X1.6 Y-2.6
X0 Y-3
X-2.1 Y-4.6
X-3.5 Y-2
X-3.9 Y-1.3
X-3.7 Y-1.9
X-1.9 Y0.4
X-2.3 Y2
X-1.6 Y1.2
X-2 Y3.6
X-2.8 Y2.8
X-3.6 Y5
X-2.2 Y2.1
X-2.9 Y0.9
X-1 Y-0.2
X-0.7 Y-0.8
X-0.1 Y-2
X2.2 Y-3.4
X3.1 Y-4
X6 Y-9.4
X3 Y-2.8
X8.7 Y-3.1
X4.2 Y-3.1
X4.8 Y-1.8
X1.9 Y-2.4
X0.3 Y-3
X-1.5 Y-2.7
X-1.9 Y-0.6
X-2.9 Y1
X-4.8 Y2.1
X-2.9 Y-0.5
X-1.9 Y-2.4
X-1.3 Y-3.8
X0.6 Y-1.9
X0.9 Y-0.6
X5.1 Y-0.1
X3.4 Y-2.3
X4.3 Y-4.3
X2.1 Y-2.3
X0.7 Y-2.9
X-0.3 Y-6.1
X1.1 Y-6
X-1 Y-6.1
X0.6 Y-2
X2.4 Y-1.9
X4.1 Y-0.3
X10 Y3
X1.6 Y1.3
X1.2 Y3.9
X0.1 Y3.2
X-0.2 Y4.2
X2.1 Y8
X-1.4 Y5.1
X-0.6 Y3
X-2 Y5.9
X-0.9 Y3
X-2 Y4.7
X-0.5 Y3.1
X0.9 Y1.8
X7.5 Y3.3
X1.3 Y1.6
X0 Y2
X-2.8 Y6.7
X-1 Y1.8
X-2.9 Y2.7
X-1.8 Y3.7
X-1.5 Y8.1
X-2.5 Y3.2
X-3 Y0.6
X-6.1 Y-0.6
X-2 Y0.7
X-1.1 Y1.7
X-0.5 Y5
X0.2 Y6.2
X-0.2 Y5.1
X1.9 Y11.6
X3.4 Y10.6
X1.1 Y6.8
X0.5 Y5.8
X1.1 Y2.9
X9 Y9.9
X4 Y2.1
X4.1 Y2
X4 Y3.5
X2.5 Y4.6
X5.8 Y5.8
X7.5 Y4
X4 Y3.3
X4 Y1.1
X6.3 Y0.8
X8.6 Y-0.6
X5.2 Y0.9
X3.6 Y2.2
X4.1 Y0.1
X8 Y-2.6
X3.7 Y-3.7
X2.5 Y-1.9
X2.9 Y-3
X4.7 Y-2.7
X2.8 Y-1.4
X5.8 Y-7.5
X1.7 Y-1.2
X1.7 Y-4
X1.1 Y-7.4
X-1.1 Y-7.8
X1.1 Y-5.3
X0 Y-5.4
X-3.8 Y-7.7
X-1.7 Y-7.4
X0.3 Y-3.2
X0.7 Y-2
X4.7 Y-4.4
X1 Y-3.1
X0.3 Y-4.2
X1.2 Y-1.7
X3.9 Y-1.9
X5.3 Y-0.1
X8.4 Y1.4
X3.8 Y-1.7
X3.1 Y-2.9
G3 X27.2 Y-12.1 I22.9 J14.9
G1 X4.9 Y2
X5.4 Y3.4
X6.2 Y2.1
X6.3 Y0.2
X12 Y-6.3
X7 Y-1.9
X14.3 Y-3
X10.6 Y-5.1
X6.2 Y-4
X3.3 Y-0.3
X3.1 Y0.5
X4.1 Y-1.1
X1.5 Y-1.4
X0.6 Y-3.9
X-0.1 Y-7.7
X-1.6 Y-7.5
X-0.9 Y-7.7
X-1.8 Y-4
X-8.1 Y-8.8
X-8.2 Y-6.1
X-7.5 Y-3.4
X-3 Y-1.3
X-2.7 Y-3.3
X-2.2 Y-3.7
X-3 Y-1.6
X-6.4 Y-0.5
X-6.6 Y1.4
X-2.1 Y-0.8
X-3.1 Y-5.6
X-2.4 Y-2.3
X-4.8 Y-7
X-0.7 Y-2.1
X0.5 Y-2
X3.5 Y-6.5
X1.5 Y-3.9
X1.4 Y-1.5
X1.9 Y-0.7
X3.2 Y0.4
X5.1 Y3.3
X12.5 Y1.2
X2.4 Y-1.9
X1.2 Y-4.1
X0 Y-4.3
X-1 Y-1.8
X-4.7 Y-2.8
X-12.8 Y-4.3
X-5.5 Y-2.3
X-5.2 Y-0.6
X-7.9 Y-3.4
X-4.1 Y-0.7
X-3 Y0.7
X-1.8 Y1.1
X-0.3 Y1
X0.8 Y1.9
X6.8 Y5.1
X2.1 Y3.7
X1.8 Y6.2
X-0.3 Y3.1
X-3.5 Y8.7
X-0.7 Y0.8
X-3.1 Y0.7
X-6.7 Y0.1
X-2.9 Y1.3
X-2.7 Y1.9
X-6.2 Y1
X-8.8 Y1
X-3.8 Y-1.6
X-5.2 Y-4.1
X-3.3 Y-2.9
X-3.6 Y-2.8
X-3.7 Y-4
X-5 Y-6.1
X-6.4 Y-9
X-2.9 Y-6.8
X-1.8 Y-1.1
X-4.4 Y-0.2
X-3.3 Y0.2
X-6.1 Y-1.7
X-4.6 Y-1.9
X-2 Y0.3
X-1.3 Y1.7
X-0.9 Y5.1
X0.6 Y4.1
X1.1 Y2.9
X0.4 Y5.1
X0.6 Y3.1
X-1.5 Y2.7
X-3.6 Y2.1
X-3.8 Y2.2
X-3.1 Y2.8
X-4.7 Y5.8
X-7.4 Y4.5
X-3.7 Y3.5
X-3.9 Y1.5
X-7.1 Y2.3
X-5.1 Y3.5
X-4.9 Y2
X-8.7 Y5.9
X-3.8 Y1.7
X-3.9 Y-0.9
X-4.3 Y-2.6
X2.8 Y-0.9
X5.1 Y-5.4
X7.2 Y-4.6
X3.3 Y-2.5
X8 Y-3
X4.2 Y-3.2
X4.4 Y-5
X4.8 Y-2.7
X3.2 Y-2.9
X3.1 Y-1.1
X5.2 Y-1.4
X2.4 Y-2.2
X2 Y-5.9
X0 Y-5.4
X-2.5 Y-9.7
X-2.3 Y-4.7
X-4.1 Y-4.5
X-1.1 Y-3
X-0.6 Y-4.3
X-5.1 Y-7.7
X-6.3 Y-1.9
X-1.3 Y-1.5
X-1.5 Y-2.6
X-2.9 Y-1.2
X-2.2 Y0.1
X-1.9 Y1
X-2.3 Y3.6
X-2 Y3.9
X-5.6 Y3.4
X-1 Y3
X-0.9 Y11.6
X-0.8 Y5.2
X-6.1 Y5.5
G3 X-7.4 Y-3.3 I-3.1 J-3
G1 X0.7 Y-1.9
X3.1 Y-2.8
X3.3 Y-2.5
X1.5 Y-2.8
X1.1 Y-6
X-1 Y-4
X4 Y-6
X1.1 Y-4.2
X1.5 Y-9.5
X-0.6 Y-5.5
X0.3 Y-4.4
X-0.6 Y-4.2
X1.2 Y-2.9
X9.1 Y-8.6
X6.2 Y-4.1
X1.1 Y-1.9
X-0.2 Y-6.4
X1.5 Y-1.5
X11.9 Y-4
X6.8 Y-2.7
X9 Y-3.1
X7 Y-5.6
X4.4 Y-1
X4.1 Y-1
X1 Y-0.5
X0.6 Y-2
X-0.4 Y-2
X-1.3 Y-1.6
X-8 Y-3.8
X-1.7 Y-1.1
X-4.4 Y0.3
X-8.5 Y0.3
X-1.8 Y-1
X-4.9 Y-6.8
X-4.9 Y-3.9
X-2.6 Y-2.1
X-4.5 Y-6.2
X-2.9 Y-1
X-3.1 Y-0.9
X-1.8 Y-2.6
X-0.7 Y-5
X-1.9 Y-3.7
X-0.1 Y-1
X1.9 Y-2.4
X5.6 Y-3
X4.8 Y-5.6
X6.1 Y-1.7
X3.1 Y-0.3
X1.4 Y-1.4
X0.7 Y-2
X-0.3 Y-3.4
X-0.6 Y-2.9
X0.9 Y-2.1
X2.4 Y-2.1
X4 Y-1.2
X6.4 Y-0.8
X6.4 Y0.7
X5.1 Y0.5
X5.5 Y-2.8
X6.3 Y-3.6
X3.1 Y-0.5
X1.8 Y0.9
X0.2 Y1
X-3.7 Y8.5
X-0.4 Y3
X0.5 Y0.9
X1.9 Y0.6
X2 Y-0.4
X6.7 Y-5.3
X3.9 Y-2.6
X3.5 Y-3
X14.7 Y-6.8
X2.9 Y-3.1
X3.6 Y-4
X5.3 Y-3.9
X2.2 Y-3.9
X1.7 Y-7.5
X0.6 Y-4.2
X2.2 Y-4.9
X2.4 Y-13.6
X1.8 Y-4.8
X0.4 Y-3.2
X0.8 Y-1.9
X-0.5 Y-3
X-0.6 Y-0.8
X-1.1 Y-0.2
X-1.6 Y2.5
X-2.1 Y7.3
X-5.9 Y9.2
X-0.6 Y4.3
X0 Y8.5
X-1.4 Y4.4
X-2.1 Y3.7
X-2.6 Y1.7
X-4.5 Y0.2
X-3.3 Y-0.8
X-1.8 Y1
X-2.1 Y3.7
X-3.1 Y2.9
X-2.9 Y1.2
X-4.2 Y-0.3
X-9.8 Y-0.3
X-4.1 Y1.4
X-7.9 Y5.7
X-2.5 Y2.2
X-6.7 Y2.5
X-5.2 Y0.5
X-3 Y-1
X-1.2 Y-1.6
X0.1 Y-2
X2.2 Y-4.9
X2.7 Y-3
X4.5 Y-2.2
X1.6 Y-2.8
X-0.1 Y-2.2
X-4 Y-3.8
X-3.1 Y-6
X-2.7 Y-1.5
X-5.3 Y-0.1
X-5.3 Y1.2
X-3.6 Y2.3
X-5 Y5.7
X-3.2 Y2.7
X-3.1 Y0.8
X-3.3 Y-0.2
X-4.7 Y-2.2
X-1.4 Y-1.5
X-1 Y-4
X0.3 Y-1
X1.8 Y-0.9
X4 Y0.3
X1.9 Y-0.8
X1.2 Y-1.6
X0.1 Y-1.1
X-1.4 Y-1.3
X-5.2 Y-1
X-2.3 Y-2.2
X-2.7 Y-5.1
X-2.5 Y-3.8
X-1.9 Y-7.4
X-1.7 Y-1.7
X-8.9 Y-6
X-5 Y-1.6
X-8.3 Y-4.4
X-11.7 Y-0.2
X-3 Y1.2
X-8.4 Y6.8
X-3.9 Y3.4
X-2 Y0.3
X-2.7 Y-1.4
X-1.4 Y-1.5
X-1.4 Y-2.7
X-1.8 Y-1.1
X-2 Y-0.1
X-1.7 Y1.1
X-0.9 Y2.9
X-0.1 Y2.1
X1.8 Y3.7
X-0.2 Y3.1
X-1.7 Y2.6
X-2.9 Y0.6
X-2.6 Y-1.5
G3 X-3.6 Y-19.5 I3.8 J-10.8
G1 X2 Y-0.7
X3.2 Y-0.1
X7.1 Y-5.9
X2.5 Y-1.9
X5.3 Y-1.4
X1.4 Y-1.4
X1.9 Y-5
X0.1 Y-2.1
X-1.1 Y-3.1
X-0.1 Y-2.1
X1 Y-1.8
X2.7 Y-1.5
X6.2 Y-0.5
X3.7 Y-1.7
X1.3 Y-1.6
X0.2 Y-1
X-1.1 Y-1.8
X-6.8 Y-3
X-3 Y-1.5
X-1.3 Y-3
X-1.2 Y-4.2
X-7.4 Y-8.4
X-5.4 Y-4
X-3.2 Y-0.7
X-3.3 Y0.3
X-4.5 Y0.5
X-6.9 Y-0.5
X-4.9 Y2.4
X-3.5 Y2.7
X-7.5 Y1.3
X-1 Y-0.4
X-2 Y-5.9
X-1.5 Y-3.8
X-1.6 Y-1.3
X-1 Y-0.2
X-1.7 Y1
X-2.9 Y8.9
X-2.9 Y4.2
X-0.3 Y1
X0.4 Y0.9
X1.9 Y0.8
X3 Y0.1
X3.1 Y-0.3
X6 Y1.6
X14.1 Y-4.2
X7.4 Y-1.7
X3.4 Y0.7
X2.1 Y1
X1.3 Y1.8
X1.6 Y3
X3.9 Y2.3
X1.7 Y2.9
X2.5 Y3.8
X1.8 Y3.8
X0.1 Y4.3
X-0.9 Y3.2
X-4.6 Y4.5
X-4.6 Y2.8
X-5.3 Y5.5
X-2 Y0.7
X-3.2 Y-0.4
X-11.9 Y-4.3
X-2.4 Y-2.4
X-2.7 Y-7.2
X-2.5 Y-1.8
X-6.8 Y-3.1
X-8.9 Y-3.8
X-12.5 Y-2
X-13.1 Y3.2
X-4.4 Y0
X-9.2 Y3.4
X-4 Y3.5
X-1.5 Y3.9
X0 Y2.1
X1.2 Y4
X-0.1 Y1.1
X-5.5 Y4.9
X-1.9 Y0.9
X-3.2 Y0.3
X-7.1 Y-1.6
X-4.9 Y-1.9
X-11.2 Y-1.9
X-2.8 Y-1.4
X-1.3 Y-1.7
X-0.8 Y-5.2
X-1.7 Y-3.8
X-0.2 Y-3.2
X-2.1 Y-2.3
X-1.3 Y-1.6
X-0.8 Y-5.1
X2.6 Y-3.3
X0.7 Y-3.1
X-0.7 Y-1.9
X-2.9 Y-2.9
X-2 Y-0.6
X-8.4 Y0.8
X-8.2 Y-1.4
X-2 Y-2.5
X-0.9 Y-2.9
X0.2 Y-1
X2.7 Y-1.4
X1.1 Y-1.7
X0 Y-1
X-2.3 Y-3.7
X-2.3 Y-3.4
X-1.9 Y-4.8
X0.5 Y-0.9
X2.1 Y-0.2
X3.1 Y1.3
X4.7 Y2.9
X7.1 Y2.2
X9.5 Y0.3
X4.6 Y2.9
X5.5 Y1
X5.4 Y-1.1
X6.1 Y-2.1
X3.9 Y-1.9
X2.8 Y-1.3
X14.5 Y-8.2
X3.7 Y-1.5
X0.6 Y-0.9
X0 Y-1
X-1.4 Y-1.6
X-3 Y-1.2
X-15.9 Y-1.8
X-3.2 Y-2.9
X-4 Y-1
X-3.1 Y0.4
X-7.1 Y1.9
X-3.1 Y2.7
X-3.7 Y1.7
X-3.7 Y3.7
X-3.8 Y1.5
X-8.4 Y-0.2
X-1.9 Y-2.3
X-1.3 Y-2.8
X-5.3 Y-3.2
X-1 Y-3
X0.7 Y-2
X7.4 Y-9.3
X15.1 Y-16.3
X22.3 Y-20.8
X20 Y-16.2
X18.4 Y-12.5
X23.7 Y-13.9
X20.6 Y-9.6
X21.2 Y-8.3
X17.3 Y-5.3
X28.1 Y-6.8
X19.8 Y-3.3
X23.3 Y-1.6
X17.5 Y-0.4
X20.2 Y0.9
X22.4 Y2.8
X18.9 Y4
X24.1 Y7.1
X31.1 Y12.1
X19.7 Y9.2
X18.1 Y10.4
X18.9 Y12.7
X18.3 Y14.4
X9.3 Y8.5
X14 Y14.7
X6.1 Y7.1
X0.8 Y3
X0 Y1
X-1.9 Y2.3
X-6.6 Y3.2
X-18.9 Y6.6
X-2.1 Y-0.4
X-6.9 Y-6.2
X-2.4 Y-2.4
X-2 Y-1
X-0.8 Y-2.1
X-0.8 Y-3.2
X-2 Y-2.5
X-6.1 Y-4.1
X-5.5 Y-4.9
X-8.2 Y-2.5
X-5 Y-1.7
X-3.2 Y0.3
X-7.1 Y1.7
X-5.4 Y0.4
X-10.3 Y2.3
X-4.4 Y2.7
X-8.3 Y1.2
X-9.3 Y-0.6
X-7.8 Y2.8
X-6 Y-0.2
X-1.8 Y1
X-0.9 Y1.7
X0.7 Y0.8
X1.9 Y0.7
X3.1 Y2.7
X7.2 Y4
X5.3 Y3.2
X1.1 Y1.7
X0.1 Y1
X-1.9 Y2.5
X-5.6 Y4.6
X-4.8 Y2.1
X-3 Y0.5
X-2.6 Y-1.7
X-1.3 Y-1.7
X-2 Y-0.5
X-2.5 Y1.7
X-2.3 Y4.6
X-2.5 Y3.2
X-0.5 Y3.1
X1.1 Y4.1
X0.9 Y3.9
X2.3 Y3.5
X1.9 Y2.5
X0.4 Y2.1
X-0.6 Y1.9
X-5.2 Y6.4
X-0.5 Y2.2
X1.1 Y1.8
X4.7 Y2.2
X2 Y3.7
X1.3 Y5.5
X2.9 Y3.1
X2.6 Y2.1
X1.8 Y4.9
X0.4 Y12.9
X0 Y3.2
X1 Y4.3
X0.6 Y4.2
X2.5 Y2
X6.2 Y4.1
X10.5 Y3.4
X10.6 Y1.4
X10.2 Y2.4
X5.9 Y4.4
X4 Y1.2
X1.1 Y-0.2
X0.8 Y-1.9
X0.5 Y-3.2
X0.8 Y-2.1
X-0.6 Y-7.4
X-0.3 Y-3.2
X3 Y-8
X0.6 Y-4.2
X-1.5 Y-4
X-1.7 Y-4
X0.3 Y-4.2
X2.8 Y-8.2
X3.8 Y-5
X1.6 Y-4
X-0.4 Y-2.9
X0.5 Y-0.9
X2.9 Y-0.6
X5.1 Y1.1
X1.8 Y-0.9
X1.3 Y-3.8
X0.4 Y-2
X4.9 Y-1.7
X2.9 Y-1.1
X8.5 Y0.6
X3.1 Y-0.6
X2.6 Y-1.8
X4.2 Y-4.9
X3.5 Y-4
X2.6 Y-6.8
X-0.4 Y-1.9
X-1.9 Y-4.7
X0 Y-1.1
X1.3 Y-1.7
X3.8 Y-1.4
X10.9 Y-3.3
X9.8 Y-3.8
X4.2 Y-0.8
X3 Y0.9
X3 Y2.9
X10 Y12.6
X9.7 Y14.5
X8.1 Y14.3
X8.6 Y17.4
X9.1 Y21.5
X5.8 Y16.5
X7.3 Y25.6
X4.1 Y19.4
X4 Y27.5
X1.1 Y21.1
X-1 Y20.2
X-3.3 Y23.3
X-6 Y33.3
X-4 Y16.2
X-6.8 Y21.1
X-9.3 Y23.3
X-10.4 Y19.9
X-8.9 Y14.3
X-10.4 Y14.7
X-0.4 Y5.3
X0.5 Y108.2
X0.2 Y38.9
X-0.3 Y29
X0.5 Y75.2
X5 Y7.4
X12.5 Y21
X7.3 Y13.4
X10.8 Y22.3
X7.8 Y18.8
X5.6 Y17.5
X5.7 Y23.2
X3.8 Y20.8
X3.4 Y30.2
X-0.9 Y28.7
X-2 Y25.7
X-3.6 Y20.7
G3 X-30 Y85.4 I-380.5 J-85.7
G1 X-8.9 Y15.8
X-12.7 Y19.5
X-11.7 Y15.2
X-10.2 Y11.3
X-1.9 Y1.2
M8
G0 X95.9 Y117.9
M7
G1 X-18 Y-9.6
X-103.6 Y2
X-8 Y0.1
X-36.7 Y0.9
X-142 Y2.9
X-18.9 Y0.4
X-74.8 Y-0.4
X-37.2 Y-0.3
X-64.6 Y-0.8
X-151.8 Y-1.4
X-3 Y-0.3
X-2.8 Y-1.7
X-1.5 Y-2.9
X-0.3 Y-11.6
X0.3 Y-56.8
X0.5 Y-127.9
X0.7 Y-63.7
X-0.2 Y-9.1
X0.4 Y-27.6
X0.3 Y-48.8
X-0.1 Y-62.7
X-1.3 Y-181.5
X0.2 Y-9
X-0.4 Y-11.5
X0.1 Y-19.8
X0 Y-6.6
X-1.2 Y-184.9
X-0.8 Y-124.8
X-0.5 Y-58.6
X0.1 Y-9
X-0.5 Y-29.8
X0.2 Y-7.8
X-0.3 Y-11.3
X-1.6 Y-192.4
X0.4 Y-8.3
X1.6 Y-2.7
X2.7 Y-1.6
X3.4 Y-0.4
X189.4 Y-3.2
X7.9 Y-0.1
X39.6 Y-0.7
X111.7 Y-1.8
X96.6 Y0.7
X4.5 Y0.4
X36 Y0.2
X179.2 Y2
X2.9 Y1.1
X2.2 Y2.3
X0.8 Y3.3
X0.2 Y207.8
X0 Y5.9
X0.1 Y33.9
X-0.2 Y25.4
X0.1 Y46.2
X0.1 Y304.3
X0.3 Y34.6
X0 Y32
X0 Y154.7
X0.6 Y112.4
X2.5 Y121
X0.8 Y39.7
X2.1 Y96.6
X0.6 Y45.2
X-1.3 Y2.8
X-3.7 Y2
X-14 Y0.7
X-17.8 Y0.3
M8
M30
```

- Visualisation Logical/Visualization (not shown)

Listed in the project but not available here: Logical/Global.typ, Logical/Global.var
